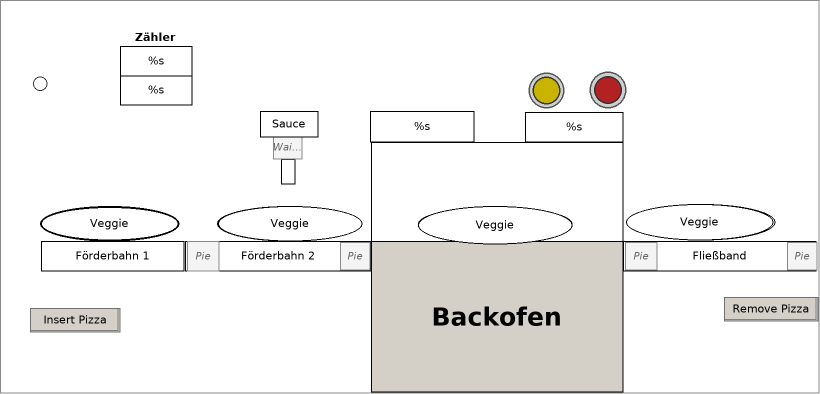
VISUALIZATION OvenHMI  // 820x394
    Rectangle (281,159 14x25), colour toggle: MAIN.veggie._zutaten MAIN.salami._zutaten
    Rectangle (185,241 186x30), "Förderbahn 2"
    Ellipse (217,206 143x35), "Salami", invisible if: NOT MAIN.salami._zutaten
    Rectangle (371,142 252x250)
    Rectangle (623,241 193x30), "Fließband"
    Ellipse (628,204 147x36), "Salami", invisible if: NOT MAIN.salami._pizza_fertig
    Button (30,308 90x24), "Insert Pizza"
        tap MAIN.Pizza_in
        OnMouseClick: execute {  }
    Button (724,297 94x24), "Remove Pizza"
        tap MAIN.Pizza_out
        OnMouseClick: execute {  }
    Ellipse (418,207 154x33), "Salami", invisible if: NOT MAIN.salami._pizza_backen
    Rectangle (371,241 252x151), "Backofen", colour toggle: MAIN.veggie._pizza_backen OR MAIN.salami._pizza_backen
    Pie (187,241 32x30)
    Pie (340,242 30x28)
    Pie (625,242 32x28)
    Pie (787,242 30x28)
    RadioButton (31,47 136x73), variable: MAIN.i
        Areas[0]: Text=Veggie
        Areas[1]: Text=Salami
    Ellipse (218,206 144x35), "Veggie", invisible if: NOT MAIN.veggie._zutaten
    Ellipse (418,206 154x38), "Veggie", invisible if: NOT MAIN.veggie._pizza_backen
    Ellipse (626,204 147x36), "Veggie", invisible if: NOT MAIN.veggie._pizza_fertig
    Rectangle (525,112 98x30), "%s", text variable: MAIN.salami.PizzaStatus, invisible if: MAIN.i=0
    Rectangle (371,112 103x30), "%s", text variable: MAIN.salami.fbTimer.ET, invisible if: MAIN.i=0
    Rectangle (120,75 72x30), "%s", text variable: MAIN.salami._count
    Rectangle (120,46 72x30), "%s", text variable: MAIN.veggie._count
    Rectangle (370,111 104x31), "%s", text variable: MAIN.veggie.fbTimer.ET, invisible if: MAIN.i=1
    Rectangle (525,112 98x30), "%s", text variable: MAIN.veggie.PizzaStatus, invisible if: MAIN.i=1
    Rectangle (41,241 143x30), "Förderbahn 1"
    Ellipse (40,206 139x35), "Salami", invisible if: NOT MAIN.salami._teig_auflade
    Lamp1 (524,70 45x41), variable: MAIN.salami._pizza_backen OR MAIN.veggie._pizza_backen, style: Lamp-Lamp1-Yellow
    Lamp1 (585,69 46x42), variable: MAIN.salami._brand_alarm OR MAIN.veggie._brand_alarm, style: Lamp-Lamp1-Red
    Ellipse (41,207 137x33), "Veggie", invisible if: NOT MAIN.veggie._teig_auflade
    WaitingSymbolFlower (273,135 29x24)
    Label (107,28 97x19), "Zähler"
    Rectangle (260,111 58x26), "Sauce"
END_VISUALIZATION

(* stored: Version 1.1.0.1, ProductVersion 3.1.4022.6
   Visu OvenHMI: Id {a2950904-96e1-441d-928f-b4716c573e07} *)
